// TwinCAT 3 PLC project PLC_FeaturePreprocessing
// ProgramVersion: 3.1.4023.0
// libraries:
//   Tc2_Standard, * (Beckhoff Automation GmbH)
//   Tc2_System, * (Beckhoff Automation GmbH)
//   Tc2_Utilities, * (Beckhoff Automation GmbH)
//   Tc3_Module, * (Beckhoff Automation GmbH)
//   Tc3_Vision, * (Beckhoff Automation GmbH)
// project tree:
//   DUTs/ E_FeatureScalingType.TcDUT, E_TransformationType.TcDUT, ST_ExtractionParams.TcDUT, ST_ScalingParams.TcDUT, ST_TransformationParams.TcDUT
//   / PlcTask.TcTTO
//   POUs/ FB_TrainingDataHandler.TcPOU, F_ExtractFeatures.TcPOU, F_GetNumberOfFeatures.TcPOU, F_VisualizeFeatures.TcPOU, MAIN.TcPOU
// real-time tasks:
//   TASK PlcTask: cycle T#40ms, priority 20, ADS port 350
//   TASK VnTask ImgAcq (TrainingImages): cycle T#10ms, priority 6, ADS port 351

CONFIGURATION PLC_FeaturePreprocessing
    RESOURCE PLC ON TwinCAT3
        TASK PlcTask(INTERVAL := T#40ms, PRIORITY := 20);
        PROGRAM MAIN WITH PlcTask : MAIN;
    END_RESOURCE
END_CONFIGURATION

// ---- DUTs/E_FeatureScalingType.TcDUT
{attribute 'qualified_only'}
{attribute 'strict'}
TYPE E_FeatureScalingType :
(
	NONE := 0,
	MAXABS,
	MINMAX,
	MINMAX_EXP,
	STANDARDIZATION,
	CUSTOM
);
END_TYPE

// ---- DUTs/E_TransformationType.TcDUT
{attribute 'qualified_only'}
{attribute 'strict'}
TYPE E_TransformationType :
(
	NONE := 0,
	PCA,
	PCA_N_Components,
	PCA_Variance,
	LDA,
	LDA_N_Components
);
END_TYPE

// ---- DUTs/ST_ExtractionParams.TcDUT
TYPE ST_ExtractionParams :
STRUCT
	bUseImageFeatures	: BOOL := TRUE; 			// If true use image features, if false use contour features
	fContourThreshold	: LREAL := 65;				// Threshold for contour extraction if active 
	ipImageWorkDisp		: ITcVnDisplayableImage;	// Image channel for feature extraction 
	ipImageBinaryDisp	: ITcVnDisplayableImage;	// Binary Image of threshold function if active
END_STRUCT
END_TYPE

// ---- DUTs/ST_ScalingParams.TcDUT
TYPE ST_ScalingParams :
STRUCT
	eScalingType	: E_FeatureScalingType;
	aCustomScaling	: ARRAY [0..18] OF LREAL := [0, 0, 0, 0, 0, 0, 0, 0, 0, 0, 0, 0, 0, 0, 0, 0, 0, 0, 0]; // The default values with 0 result in no scaling, for custom scaling please enter valid values.
END_STRUCT
END_TYPE

// ---- DUTs/ST_TransformationParams.TcDUT
TYPE ST_TransformationParams :
STRUCT
	eTransformType			: E_TransformationType;
	nPcaComponentNum		: UDINT := 2;
	fPcaRetainedVariance	: LREAL := 0.95;
	nLdaComponentNum		: UDINT := 1;
END_STRUCT
END_TYPE

// ---- POUs/MAIN.TcPOU
PROGRAM MAIN
VAR
	stExtractionParams		:	ST_ExtractionParams;	// Feature extraction options
	stScalingParams			:	ST_ScalingParams;		// Feature scaling type and custom values
	stTransformationParams	:	ST_TransformationParams;// Transformation type and parameters
	
	bResetTrainingData		:	BOOL;					// Reset the sample features to get new onces
	bResetScaling			:	BOOL;					// Reset the feature scaling to get new onces and visualize the result
	bResetModel				:	BOOL;					// Reset model to start a new transformation with a changed model or parameters
	nSelectedFeatureID		:	UDINT;					// ID of the feature in the vector that should be visualized
	bVisualizeFeatures		:	BOOL;					// Create new feature visualization image
	
	hr						:	HRESULT;
	hrLastExecution			:	HRESULT;
	ipImageResDisp			:	ITcVnDisplayableImage;
	fbTrainingDataHandler	:	FB_TrainingDataHandler;

	ipTransformationModel	:	ITcVnMlModel;
	ipSamplesTraining		:	ITcVnContainer;
	ipClassLabels			:	ITcVnContainer;
	ipFeatureScaling		:	ITcVnContainer;
	ipScaledSamples			:	ITcVnContainer;
	ipTransformedSamples	:	ITcVnContainer;
	
	nNumberOfSamples		:	ULINT;
	nNumberOfFeatures		:	ULINT;
	nNumberOfCustomScales	:	ULINT;
END_VAR

// Disclaimer

// This publication contains statements about the suitability of our products for certain
// areas of application. These statements are based on typical features of our products.
// The examples shown in this publication are for demonstration purposes only.
// The information provided herein should not be regarded as specific operation characteristics.
// It is incumbent on the customer to check and decide whether a product is suitable for use
// in a particular application. We do not give any warranty that the source code which is
// made available with this publication is complete or accurate.

// THE SAMPLE CODE CONTAINED IN THIS PUBLICATION IS PROVIDED “AS IS” WITHOUT WARRANTY OF ANY KIND,
// EITHER EXPRESSED, IMPLIED OR STATUTORY, INCLUDING WITHOUT LIMITATION, ANY WARRANTY WITH RESPECT TO NON-INFRINGEMENT,
// FREEDOM FROM PROPRIETARY RIGHTS OF THIRD PARTIES OR FITNESS FOR ANY PARTICULAR PURPOSE.

// This publication may be changed from time to time without prior notice.
// No liability is assumed for errors and/or omissions.
// Our products are described in detail in our data sheets and documentations.
// Product-specific warnings and cautions must be observed.
// For the latest version of our data sheets and documentations visit our website (www.beckhoff.de).

// © Beckhoff Automation GmbH & Co. KG, June 2023

// The reproduction, distribution and utilization of this document as well as the communication
// of its contents to others without express authorization is prohibited. 
// Offenders will be held liable for the payment of damages.
// All rights reserved in the event of the grant of a patent, utility model or design.

//	==========================================================================================

// SAMPLE - Machine Learning Feature Preprocessing
//	-------------------------------------------------------

// Steps To Do:
// ------------
// 1. Add the training images to the TrainingImages control
// 2. Activate the configuration -> Start TwinCAT system and PLC to run -> see the result in the ADS Image Watch
// 3. Change stExtractionParams to change the feature that are extraced by F_ExtractFeatures or the function parameters
// 4. Change stScalingParams or stTransformationParams to change the feature scaling or the transformation model
// 5. Set bResetTrainingData to get new training data if images or feature extraction changed
// 6. Set bResetScaling to get new feature scaling if stScalingParams changed
// 7. Set bResetModel to get new transformation model if the model type or parameters changed
// 8. Set nSelectedFeatureID to a feature index that should bei visualized
// 9. Set bVisualizeFeatures to update the visualization image

// Reset return value
hr := S_OK;

// Reset the trained features to get new ones
IF bResetTrainingData THEN
	bResetTrainingData := FALSE;
	bVisualizeFeatures := TRUE;
	fbTrainingDataHandler.Reset();
	FW_SafeRelease(ADR(ipSamplesTraining));
	FW_SafeRelease(ADR(ipClassLabels));
	FW_SafeRelease(ADR(ipFeatureScaling));
	FW_SafeRelease(ADR(ipScaledSamples));
	FW_SafeRelease(ADR(ipTransformationModel));
END_IF

// Get sample data for feature preprocessing
fbTrainingDataHandler(stExtractionParams := stExtractionParams);
IF ipSamplesTraining = 0 AND ipClassLabels = 0 THEN
	hr := fbTrainingDataHandler.GetTrainingData(ipSamplesTraining, ipClassLabels);
END_IF

// Reset to get new scaling with changed type or parameters
IF bResetScaling THEN
	bResetScaling := FALSE;
	bVisualizeFeatures := TRUE;
	FW_SafeRelease(ADR(ipFeatureScaling));
	FW_SafeRelease(ADR(ipScaledSamples));
	FW_SafeRelease(ADR(ipTransformationModel));
END_IF

// Feature scaling
IF SUCCEEDED(hr) AND ipSamplesTraining <> 0 AND ipScaledSamples = 0 THEN
	// Get or create scaling
	CASE stScalingParams.eScalingType OF
		E_FeatureScalingType.MAXABS:
			hr := F_VN_GetFeatureScales(ipSamplesTraining, ipFeatureScaling, TCVN_FST1_MAXABS, hr);
			
		E_FeatureScalingType.MINMAX, E_FeatureScalingType.MINMAX_EXP:
			hr := F_VN_GetFeatureScales(ipSamplesTraining, ipFeatureScaling, TCVN_FST1_MINMAX, hr);
			
		E_FeatureScalingType.STANDARDIZATION:
			hr := F_VN_GetFeatureScales(ipSamplesTraining, ipFeatureScaling, TCVN_FST1_STANDARDIZATION, hr);
			
		E_FeatureScalingType.CUSTOM:
			// Structure of the scaling container
			// The first element of the ipScales container contains the value of ETcVnFeatureScalingType.
			// For MAXABS this is followed by 1 positive scaling value per feature to get scaled values between [-1..1].
			// For MINMAX and STANDARDIZATION there are 2 scaling values per feature.
			// For MINMAX the min and max values follow for each feature to get scaled values between [0..1].
			// For STANDARDIZATION the mean and standard deviations values follow for each feature to get scaled values wih mean = 0 and std = 1.
			
			// Custom scaling
			// To create a custom scaling first the eFeatureScalingType must be written into the stScalingParams.aCustomScaling[0] of the array.
			// After that the other array elements must be filled according to the chosen scaling type.
			// Finally select the stScalingParams.eScalingType = CUSTOM and start the creation of the custom scaling with bResetScaling.
			
			// Get the number of samples and features
			hr := F_GetNumberOfFeatures(ipTransformedSamples, nNumberOfSamples, nNumberOfFeatures, hr);
			
			// Check the scaling type and compare the array length with the number of features 
			CASE LREAL_TO_DINT(stScalingParams.aCustomScaling[0]) OF
				
				TCVN_FST1_MAXABS:
					IF SIZEOF(stScalingParams.aCustomScaling) / SIZEOF(LREAL) < nNumberOfFeatures + 1 THEN
						hr := Tc2_System.E_HRESULTAdsErr.INVALIDSIZE;
					ELSE
						nNumberOfCustomScales := nNumberOfFeatures + 1;
					END_IF
					
				TCVN_FST1_MINMAX, TCVN_FST1_STANDARDIZATION:
					IF SIZEOF(stScalingParams.aCustomScaling) / SIZEOF(LREAL) < (nNumberOfFeatures * 2) + 1 THEN
						hr := Tc2_System.E_HRESULTAdsErr.INVALIDSIZE;
					ELSE
						nNumberOfCustomScales := (nNumberOfFeatures * 2) + 1;
					END_IF
			ELSE
				hr := Tc2_System.E_HRESULTAdsErr.INVALIDPARM;
			END_CASE

			// Create container with custom scaling values
			hr := F_VN_CreateContainerFromArray(ADR(stScalingParams.aCustomScaling), ipFeatureScaling, ContainerType_Vector_LREAL, nNumberOfCustomScales, hr);
	END_CASE

	IF stScalingParams.eScalingType = E_FeatureScalingType.NONE THEN
		// Copy container for no scaling
		FW_SafeRelease(ADR(ipScaledSamples));
		hr := F_VN_CopyContainer(ipSamplesTraining, ipScaledSamples, hr);
		
	ELSIF stScalingParams.eScalingType = E_FeatureScalingType.MINMAX_EXP THEN
		// Apply scaling with custom output range
		hr := F_VN_FeatureScalingExp(ipSamplesTraining, ipFeatureScaling, ipScaledSamples, 0.1, 0.9, hr);
	ELSE
		// Apply scaling
		hr := F_VN_FeatureScaling(ipSamplesTraining, ipFeatureScaling, ipScaledSamples, hr);
	END_IF
	
	hrLastExecution := hr;
	bVisualizeFeatures := TRUE;
END_IF

// Retrain with changed model or parameters
IF bResetModel THEN
	bResetModel := FALSE;
	bVisualizeFeatures := TRUE;
	FW_SafeRelease(ADR(ipTransformationModel));
END_IF

// Feature transformation model
// Note: For LDA-based feature transformation, the number of training samples must be greater than or equal to the number of features.
IF SUCCEEDED(hr) AND stTransformationParams.eTransformType > E_TransformationType.NONE AND ipScaledSamples <> 0 AND ipTransformationModel = 0 THEN
	// Create the model
	CASE stTransformationParams.eTransformType OF	
		E_TransformationType.PCA:
			hr := F_VN_CreatePcaTransform(ipTransformationModel, ipScaledSamples, hr);
			
		E_TransformationType.PCA_N_Components:
			hr := F_VN_CreatePcaTransformViaComponentNum(ipTransformationModel, ipScaledSamples, stTransformationParams.nPcaComponentNum, hr);
			
		E_TransformationType.PCA_VARIANCE:
			hr := F_VN_CreatePcaTransformViaVariance(ipTransformationModel, ipScaledSamples, stTransformationParams.fPcaRetainedVariance, hr);
			
		E_TransformationType.LDA:
			hr := F_VN_CreateLdaTransform(ipTransformationModel, ipScaledSamples, ipClassLabels, hr);
			
		E_TransformationType.LDA_N_Components:
			hr := F_VN_CreateLdaTransformViaComponentNum(ipTransformationModel, ipScaledSamples, ipClassLabels, stTransformationParams.nLdaComponentNum, hr);
	END_CASE;
	
	hrLastExecution := hr;
	bVisualizeFeatures := TRUE;
END_IF

// Feature transformation and visualization
IF SUCCEEDED(hr) AND ipScaledSamples <> 0 AND bVisualizeFeatures THEN
	bVisualizeFeatures := FALSE;
	
	IF stTransformationParams.eTransformType = E_TransformationType.NONE THEN
		// Copy container for no transformation
		FW_SafeRelease(ADR(ipTransformedSamples));
		hr := F_VN_CopyContainer(ipScaledSamples, ipTransformedSamples, hr);
	ELSE
		// Execute the feature transformation
		hr := F_VN_FeatureTransform(ipTransformationModel, ipScaledSamples, ADR(ipTransformedSamples), hr);
	END_IF

	// Get the number of samples and features
	hr := F_GetNumberOfFeatures(ipTransformedSamples, nNumberOfSamples, nNumberOfFeatures, hr);
	// Limit the ID to valid number
	nSelectedFeatureID := MIN(nSelectedFeatureID, ULINT_TO_UDINT(nNumberOfFeatures - 1));
		
	// Create a visualization image
	hr := F_VisualizeFeatures(ipTransformedSamples, nSelectedFeatureID, ipClassLabels, 600, 300, ipImageResDisp, hr);
	hrLastExecution := hr;
END_IF

END_PROGRAM

// ---- POUs/FB_TrainingDataHandler.TcPOU
FUNCTION_BLOCK PUBLIC FB_TrainingDataHandler
VAR_INPUT
	stExtractionParams		:	REFERENCE TO ST_ExtractionParams;
END_VAR
VAR_OUTPUT
END_VAR
VAR
	hr						: HRESULT;
	eCameraState			: ETcVnCameraState;
	fbCameraTraining		: FB_VN_SimpleCameraControl;	
	ipImageTraining			: ITcVnImage;
	ipImageTrainingDisp		: ITcVnDisplayableImage;
	bTrigger				: BOOL := TRUE;
	sLabel					: STRING(255);
	aGreen					: TcVnVector4_LREAL := [0, 255, 0];
	
	// Image Info
	nImagesTotal			: UDINT := 12;
	nImagesLoaded			: UDINT := 0;
	
	ipFeatures				: ITcVnContainer;
	ipImageFeatures			: ITcVnContainer;
	ipLabels				: ITcVnContainer;
END_VAR

// Initialize container
IF ipImageFeatures = 0 THEN
	hr := F_VN_CreateContainer(ipImageFeatures, ContainerType_Vector_Vector_LREAL, nImagesTotal, hr);
	hr := F_VN_CreateContainer(ipLabels, ContainerType_Vector_DINT, nImagesTotal, hr);
END_IF

// Get training images
eCameraState := fbCameraTraining.GetState();

IF eCameraState = TCVN_CS_ERROR THEN
	hr := fbCameraTraining.Reset();
	
// Camera trigger image
ELSIF eCameraState = TCVN_CS_TRIGGERING THEN
	hr := fbCameraTraining.TriggerImage();
	
ELSIF eCameraState < TCVN_CS_ACQUIRING THEN
	hr := fbCameraTraining.StartAcquisition();

// Camera streaming
ELSIF eCameraState = TCVN_CS_ACQUIRING THEN

	IF bTrigger THEN
		hr := fbCameraTraining.TriggerImage();
		IF SUCCEEDED(hr) THEN
			bTrigger := FALSE;
		END_IF
	ELSE
		hr := fbCameraTraining.GetCurrentImage(ipImageTraining);

		// Check if new image was received
		IF SUCCEEDED(hr) AND ipImageTraining <> 0 THEN
			
			// Get features from training image 
			hr := F_ExtractFeatures(stExtractionParams, ipImageTraining, ipFeatures, hr);
		
			// Add features and label to the containers. First class label = 0, second class = 1
			hr := F_VN_SetAt_ITcVnContainer(ipFeatures, ipImageFeatures, nImagesLoaded, hr);
			FW_SafeRelease(ADR(ipFeatures));
			hr := F_VN_SetAt_DINT(UDINT_TO_DINT(nImagesLoaded / 6), ipLabels, nImagesLoaded, hr);
			
			// Display image
			sLabel := CONCAT('Image Number: ', UDINT_TO_STRING(nImagesLoaded + 1));
			hr := F_VN_PutTextExp(sLabel, ipImageTraining, 30, 60, TCVN_FT_HERSHEY_PLAIN, 4, aGreen, 2, TCVN_LT_ANTIALIASED, FALSE, hr);
			hr := F_VN_TransformIntoDisplayableImage(ipImageTraining, ipImageTrainingDisp, hr);
			
			nImagesLoaded := nImagesLoaded + 1;
			IF nImagesLoaded < nImagesTotal THEN
				// Trigger next image
				bTrigger := TRUE;
			END_IF
		END_IF
	END_IF
END_IF

METHOD PUBLIC GetTrainingData : HRESULT
VAR_INPUT
	ipTrainingSamples	: REFERENCE TO ITcVnContainer;
	ipClassLabels		: REFERENCE TO ITcVnContainer;
END_VAR
VAR
	hr					: HRESULT;
END_VAR
IF nImagesLoaded = nImagesTotal THEN
	hr := F_VN_CopyContainer(ipImageFeatures, ipTrainingSamples, hr);
	GetTrainingData := F_VN_CopyContainer(ipLabels, ipClassLabels, hr);
ELSE
	GetTrainingData := S_PENDING;
END_IF
END_METHOD

METHOD PUBLIC Reset : HRESULT
VAR_INPUT
END_VAR
nImagesLoaded := 0;
FW_SafeRelease(ADR(ipFeatures));
FW_SafeRelease(ADR(ipImageFeatures));
FW_SafeRelease(ADR(ipLabels));
bTrigger := TRUE;
END_METHOD

END_FUNCTION_BLOCK

// ---- POUs/F_ExtractFeatures.TcPOU
FUNCTION F_ExtractFeatures : HRESULT
VAR_INPUT
	stExtractionParams	:	REFERENCE TO ST_ExtractionParams;
	ipImage				:	ITcVnImage;
	ipFeatures			:	REFERENCE TO ITcVnContainer;
	hrPrev				:	HRESULT;
END_VAR
VAR
	hr					:	HRESULT;
	stImageInfo			:	TcVnImageInfo;
	fChannelSize		:	LREAL;
	ipImageWork 		:	ITcVnImage;
	aAverage			:	TcVnVector4_LREAL;
	stMoments			:	TcVnMoments;
	ipDestHistogram		:	ITcVnContainer;
	nBins				:	UDINT := 4;
	fLowerBound			:	LREAL := 0;
	fUpperBound			:	LREAL := 256;
	ipHistChannel		:	ITcVnContainer;
	nElement			:	UDINT;
	ipImageBinary		:	ITcVnImage;
	ipContourList		:	ITcVnContainer;
	ipContour			:	ITcVnContainer;
	ipIterator			:	ITcVnForwardIterator;
	fArea				:	LREAL;
	fMaxArea			:	LREAL;
	nIndex				:	ULINT;
	i					:	ULINT;
	fCircularity		:	LREAL;
	fConvexity			:	LREAL;
	fPerimeter			:	LREAL;
	fInertiaRatio		:	LREAL;
	aHuInvariants		:	TcVnArray7_LREAL;
	stRectangle			:	TcVnRotatedRectangle;
END_VAR

IF FAILED(hrPrev) THEN
	F_ExtractFeatures := hrPrev;
	RETURN;
END_IF

IF ipImage = 0 THEN
	F_ExtractFeatures := Tc2_System.E_HRESULTAdsErr.INVALIDPARM;
	RETURN;
END_IF

// Convert image from RGB to Gray if nessesary
hr := F_VN_GetImageInfo(ipImage, stImageInfo, hr); 
IF stImageInfo.stPixelFormat.nChannels = 3 AND stImageInfo.stPixelFormat.ePixelEncoding = TCVN_PE_NONE THEN
	hr := F_VN_GetImageChannel(ipImage, ipImageWork, 0, hr);
	fChannelSize := ULINT_TO_LREAL(stImageInfo.nImageSize) / 3;
ELSE
	ipImageWork := ipImage;
	fChannelSize := ULINT_TO_LREAL(stImageInfo.nImageSize);
	ipImage.TcAddRef();
END_IF

// Create feature vector container
hr := F_VN_CreateContainer(ipFeatures, ContainerType_VECTOR_LREAL, 0, hr);

// *** Image features ******************************************************************************
IF stExtractionParams.bUseImageFeatures THEN
	// Average intensity
	hr := F_VN_ImageAverage(ipImage, aAverage, hr);
	hr := F_VN_AppendToContainer_LREAL(aAverage[0], ipFeatures, hr);
	hr := F_VN_AppendToContainer_LREAL(aAverage[1], ipFeatures, hr);
	hr := F_VN_AppendToContainer_LREAL(aAverage[2], ipFeatures, hr);
	
	// Image moments
	hr := F_VN_ImageMoments(ipImageWork, stMoments, FALSE, hr);
	hr := F_VN_AppendToContainer_LREAL(stMoments.fMu02, ipFeatures, hr);
	hr := F_VN_AppendToContainer_LREAL(stMoments.fMu20, ipFeatures, hr);
	
	// Histogramm 
	hr := F_VN_HistogramExp(ipImage, ipDestHistogram, nBins, fLowerBound, fUpperBound, 0, hr);
	// Get result of the first channel and scale with image size
	hr := F_VN_GetAt_ITcVnContainer(ipDestHistogram, ipHistChannel, 0, hr);
	hr := F_VN_GetAt_UDINT(ipHistChannel, nElement, 0, hr);
	hr := F_VN_AppendToContainer_LREAL(UDINT_TO_LREAL(nElement) / fChannelSize, ipFeatures, hr);
	hr := F_VN_GetAt_UDINT(ipHistChannel, nElement, 1, hr);
	hr := F_VN_AppendToContainer_LREAL(UDINT_TO_LREAL(nElement) / fChannelSize, ipFeatures, hr);
	hr := F_VN_GetAt_UDINT(ipHistChannel, nElement, 2, hr);
	hr := F_VN_AppendToContainer_LREAL(UDINT_TO_LREAL(nElement) / fChannelSize, ipFeatures, hr);
	hr := F_VN_GetAt_UDINT(ipHistChannel, nElement, 3, hr);
	hr := F_VN_AppendToContainer_LREAL(UDINT_TO_LREAL(nElement) / fChannelSize, ipFeatures, hr);
	
ELSE
// *** Contour features ****************************************************************************
	hr := F_VN_Threshold(ipImageWork, ipImageBinary, stExtractionParams.fContourThreshold, 255, ETcVnThresholdType.TCVN_TT_BINARY, hr);
	hr := F_VN_FindContours(ipImageBinary, ipContourList, hr);
	hr := F_VN_TransformIntoDisplayableImage(ipImageBinary, stExtractionParams.ipImageBinaryDisp, S_OK);
	
	// Find the largest contour in the image
	hr := F_VN_GetForwardIterator(ipContourList, ipIterator, hr);
	WHILE SUCCEEDED(hr) AND_THEN ipIterator.CheckIfEnd() <> S_OK DO
		hr := F_VN_GetContainerExp(ipIterator, ipContour, 1, hr);
	
		hr := F_VN_ContourArea(ipContour, fArea, hr);
		IF fArea > fMaxArea THEN
			// Get the value and index of the largest contour
			fMaxArea := fArea;
			nIndex := i;
		END_IF
		i := i + 1;
	END_WHILE
	
	// Area
	hr := F_VN_AppendToContainer_LREAL(fMaxArea, ipFeatures, hr);
	
	// Get container with the largest contour
	hr := F_VN_GetAt_ITcVnContainer(ipContourList, ipContour, nIndex, hr);
	
	// Circularity
	hr := F_VN_ContourCircularity(ipContour, fCircularity, hr);
	hr := F_VN_AppendToContainer_LREAL(fCircularity, ipFeatures, hr);
	
	// Convexity
	hr := F_VN_ContourConvexity(ipContour, fConvexity, hr);
	hr := F_VN_AppendToContainer_LREAL(fConvexity, ipFeatures, hr);
	
	// Perimeter
	hr := F_VN_ContourPerimeter(ipContour, fPerimeter, FALSE, hr);
	hr := F_VN_AppendToContainer_LREAL(fPerimeter, ipFeatures, hr);
	
	// Contour moment invariants
	hr := F_VN_ContourMoments(ipContour, stMoments, hr);
	hr := F_VN_HuMomentInvariants(stMoments, aHuInvariants, hr);
	hr := F_VN_AppendToContainer_LREAL(aHuInvariants[0], ipFeatures, hr);
	hr := F_VN_AppendToContainer_LREAL(aHuInvariants[1], ipFeatures, hr);
	
	// Object width and height
	hr := F_VN_EnclosingRectangle(ipContour, stRectangle, hr);
	hr := F_VN_AppendToContainer_LREAL(stRectangle.stSize.fWidth, ipFeatures, hr);
	hr := F_VN_AppendToContainer_LREAL(stRectangle.stSize.fHeight, ipFeatures, hr);
END_IF

// Release interface pointer
hr := F_VN_TransformIntoDisplayableImage(ipImageWork, stExtractionParams.ipImageWorkDisp, S_OK);
FW_SafeRelease(ADR(ipImageWork));
FW_SafeRelease(ADR(ipImageBinary));
FW_SafeRelease(ADR(ipDestHistogram));
FW_SafeRelease(ADR(ipHistChannel));
FW_SafeRelease(ADR(ipContourList));
FW_SafeRelease(ADR(ipContour));
FW_SafeRelease(ADR(ipIterator));

F_ExtractFeatures := hr;

END_FUNCTION

// ---- POUs/F_GetNumberOfFeatures.TcPOU
FUNCTION F_GetNumberOfFeatures : HRESULT
VAR_INPUT
	ipContainerList		:	ITcVnContainer;
	nNumberOfSamples	:	REFERENCE TO ULINT;
	nNumberOfFeatures	:	REFERENCE TO ULINT;
	hrPrev				:	HRESULT;
END_VAR
VAR
	hr					:	HRESULT;
	ipContainer			:	ITcVnContainer;
END_VAR

IF FAILED(hrPrev) THEN
	F_GetNumberOfFeatures := hrPrev;
	RETURN;
END_IF

IF ipContainerList = 0 THEN
	F_GetNumberOfFeatures := Tc2_System.E_HRESULTAdsErr.INVALIDPARM;
	RETURN;
END_IF

IF ipContainerList.CheckIfBasicContainer() = S_OK THEN
	F_GetNumberOfFeatures := Tc2_System.E_HRESULTAdsErr.INVALIDPARM;
	RETURN;
END_IF

// Get the number of samples
hr := F_VN_GetNumberOfElements(ipContainerList, nNumberOfSamples, hr);
IF nNumberOfSamples >= 1 THEN
	hr := F_VN_GetAt_ITcVnContainer(ipContainerList, ipContainer, 0, hr);
	// Get the number of features
	hr := F_VN_GetNumberOfElements(ipContainer, nNumberOfFeatures, hr);
END_IF

FW_SafeRelease(ADR(ipContainer));
F_GetNumberOfFeatures := hr;

END_FUNCTION

// ---- POUs/F_VisualizeFeatures.TcPOU
(* Visualize one selected feature from a sample vector in a bar chart *)
FUNCTION F_VisualizeFeatures : HRESULT
VAR_INPUT
	ipSamplesTraining	: ITcVnContainer;
	nFeatureID			: UDINT;
	ipLabels			: ITcVnContainer;
	nDestImageWidth		: UDINT := 900;
	nDestImageHeight	: UDINT := 600;
	ipDestImageDisp		: REFERENCE TO ITcVnDisplayableImage;
	hrPrev				: HRESULT;
END_VAR
VAR
	hr					: HRESULT;
	ipChartImage		: ITcVnImage;
	ipIterator			: ITcVnForwardIterator;
	ipSample			: ITcVnContainer;
	ipFeatureVector		: ITcVnContainer;
	nNumberOfSamples	: ULINT;
	nNumberOfFeatures	: ULINT;
	fValue				: LREAL;
	fMax				: LREAL;
	fMin				: LREAL;
	fScale				: LREAL;
	nOffsetX			: UDINT := 20;
	nOffsetY			: UDINT;
	fGapRatio			: LREAL := 0.25;
	nBarGapWidth		: UDINT;
	nBarWidth			: UDINT;
	i					: ULINT;
	nBarHeight			: UDINT;
	nLabelID			: DINT;
	stRectangle			: TcVnRectangle_UDINT;
	nValuePositionY		: UDINT;
	nIndexPositionY		: UDINT;
	stext				: STRING;
	
	aColorBlack			: TcVnVector4_LREAL := [0, 0, 0];
	aColorWhite			: TcVnVector4_LREAL := [255, 255, 255];
	// Colors to visualize the feature data if ipClassLabels are available. 
	// Note: Add more colors if you have more classes. 
	aColorPalette		: ARRAY [0..7]  OF TcVnVector4_LREAL :=[[255, 100, 100, 255],	// Class Label 1
																[100, 255, 100, 255],	// Class Label 2
																[100, 100, 255, 255],	// Class Label 3
																[255, 255, 100, 255],	// Class Label 4
																[100, 255, 255, 255],	// Class Label 5
																[ 10, 125, 255, 255],	// Class Label 6
																[125, 125, 125, 255],	// Class Label 7
																[255, 255, 255, 255]];	// Class Label 8

END_VAR

IF FAILED(hrPrev) THEN
	F_VisualizeFeatures := hrPrev;
	RETURN;
END_IF

IF ipSamplesTraining = 0 THEN
	F_VisualizeFeatures := Tc2_System.E_HRESULTAdsErr.INVALIDPARM;
	RETURN;
END_IF

// Get the number of samples
hr := F_VN_GetNumberOfElements(ipSamplesTraining, nNumberOfSamples, hr);
IF nNumberOfSamples = 0 THEN
	F_VisualizeFeatures := Tc2_System.E_HRESULTAdsErr.INVALIDPARM;
	RETURN;
END_IF
	
// Extract the feature vector (Vector_LREAL) from ipSamplesTraining (Vector_Vector_LREAL)
hr := F_VN_GetForwardIterator(ipSamplesTraining, ipIterator, hr);
hr := F_VN_CreateContainer(ipFeatureVector, ContainerType_Vector_LREAL, 0, hr);

WHILE SUCCEEDED(hr) AND_THEN ipIterator.CheckIfEnd() <> S_OK DO
	hr := F_VN_GetContainerExp(ipIterator, ipSample, 1, hr);
	
	hr := F_VN_GetNumberOfElements(ipSample, nNumberOfFeatures, hr);
	IF nNumberOfFeatures = 0 OR nFeatureID > nNumberOfFeatures -1 THEN
		F_VisualizeFeatures := Tc2_System.E_HRESULTAdsErr.INVALIDPARM;
		RETURN;
	END_IF
	
	// Get the requested feature and add it to the result vector  
	hr := F_VN_GetAt_LREAL(ipSample, fValue, nFeatureID, hr);
	hr := F_VN_AppendToContainer_LREAL(fValue, ipFeatureVector, hr);
END_WHILE

FW_SafeRelease(ADR(ipSample));
FW_SafeRelease(ADR(ipIterator));

// Determine the scaling for the visualization since only positive values can be displayed in the result image
hr := F_VN_MaxElementElementwise_LREAL(ipFeatureVector, fMax, hr);
hr := F_VN_MinElementElementwise_LREAL(ipFeatureVector, fMin, hr);

IF fMax < ABS(fMin) THEN
	fMax := ABS(fMin);
END_IF

// Calulate scales
fScale := (nDestImageHeight - 2 * nOffsetX) / (2 * fMax);
nBarGapWidth := TO_UDINT((nDestImageWidth - 2 * nOffsetX) / nNumberOfSamples);
nBarWidth := TO_UDINT((1 - fGapRatio) * nBarGapWidth);
nOffsetY := nDestImageHeight / 2;

// Create result image chart
hr := F_VN_CreateImageAndSetPixels(ipChartImage, nDestImageWidth, nDestImageHeight, TCVN_ET_USINT, 3, aColorWhite, hr);

FOR i := 0 TO nNumberOfSamples - 1 DO
	hr := F_VN_GetAt_LREAL(ipFeatureVector, fValue, i, hr);
	nBarHeight := LREAL_TO_UDINT(ABS(fValue * fScale));
	
	// Show the features with different colors according to the label, if labels are available
	IF ipLabels <> 0 THEN
		hr := F_VN_GetAt_DINT(ipLabels, nLabelID, i, hr);
		// Check that the class number is not larger than the aColorPalette entries
		IF nLabelID > 7 THEN
			F_VisualizeFeatures := Tc2_System.E_HRESULTAdsErr.INVALIDSIZE;
			RETURN;
		END_IF
	ELSE	
		nLabelID := 0;
	END_IF
	
	// Calulate the values of the bar
	stRectangle.nX := nOffsetX + ULINT_TO_UDINT(i) * (nBarWidth + LREAL_TO_UDINT(fGapRatio * nBarGapWidth));
	stRectangle.nY := nOffsetY  - nBarHeight;
	stRectangle.nWidth := nBarWidth;
	stRectangle.nHeight := nBarHeight;
	
	// Calculate different Y positions for negative values 
	IF(fValue < 0) THEN
		stRectangle.nY := nOffsetY;
		nValuePositionY := nOffsetY + nBarHeight + 10;
		nIndexPositionY := stRectangle.nY - 4;
	ELSE
		nValuePositionY := stRectangle.nY - 4;
		nIndexPositionY := nOffsetY + 10;
	END_IF
	
	// Draw the bar
	hr := F_VN_DrawRectangle_TcVnRectangle_UDINT(stRectangle, ipChartImage, aColorPalette[nLabelID], -1, hr);
	
	// Draw the value label
	IF ABS(fValue) < 0.1 THEN
		stext := LREAL_TO_FMTSTR(fValue, 3, FALSE);
	ELSIF ABS(fValue) < 10.0 THEN
		stext := LREAL_TO_FMTSTR(fValue, 2, FALSE);
	ELSE
		stext := LREAL_TO_FMTSTR(fValue, 1, FALSE);
	END_IF	
	hr := F_VN_PutLabelExp(stext, ipChartImage, stRectangle.nX, nValuePositionY, 0.3, 1, TCVN_FT_HERSHEY_SIMPLEX, aColorBlack, aColorWhite, TCVN_LT_8_CONNECTED, hr);
	
	// Draw the feature indexes label
	stext := ULINT_TO_STRING(i);
	hr := F_VN_PutLabelExp(stext, ipChartImage, stRectangle.nX, nIndexPositionY, 0.3, 1, TCVN_FT_HERSHEY_SIMPLEX, aColorBlack, aColorWhite, TCVN_LT_8_CONNECTED, hr);
	
END_FOR

// Draw the X-Axis line
hr := F_VN_DrawLine(nOffsetX, nOffsetY, nDestImageWidth - nOffsetX, nOffsetY, ipChartImage, aColorBlack, 1, hr);

// Draw a border around the chart
hr := F_VN_DrawRectangle(0, 0, nDestImageWidth - 1, nDestImageHeight - 1, ipChartImage, aColorBlack, 1, hr);

// Display result bar chart
hr := F_VN_TransformIntoDisplayableImage(ipChartImage, ipDestImageDisp, S_OK);

FW_SafeRelease(ADR(ipFeatureVector));
F_VisualizeFeatures := hr;

END_FUNCTION
